FUNCTION_BLOCK Test_TimestampAsFilenameString EXTENDS TUnitTestBase
VAR
    TimeStruct : TIMESTRUCT := (wDay := 23, wMonth := 12, wYear := 1945, wHour := 22, wMinute := 20, wSecond := 18, wMilliseconds := 512);
END_VAR

Assertion.AssertEquals_STRING(
    Expected := '1945-12-23 22-20-18',
    Actual   := F_TimestampAsFilenameString(TimeStruct),
    ObjectName := _TestName,
    VariableName  := 'F_TimeAsString_ms(TimeStruct)');


Test_Finished();

END_FUNCTION_BLOCK

(* stored: Version 1.1.0.1, ProductVersion 3.1.4024.3
   POU Test_TimestampAsFilenameString: Id {be314818-0935-0ff5-2754-1e6cba9ef99d}, SpecialFunc None *)
